// function block for inductive sensor with the option of debouncing + rising and falling edge detection.
FUNCTION_BLOCK FB_InductiveSensor IMPLEMENTS  I_Component
VAR_INPUT
	bSignal			: BOOL;		// Raw input sensor
	tDebounce		: TIME;		// Debounce time
// Interface vars
	sName			: STRING[20];
	bEnable     	: BOOL;
	bStart      	: BOOL;
	bHalt			: BOOL;
	bStop       	: BOOL;
	eMode       	: E_ComponentMode; 		// 0=OFF, 1=AUTO, 2=MANUAL	
END_VAR

VAR_OUTPUT
	bActive			: BOOL;
	bRising			: BOOL;
	bFalling		: BOOL;
// interface vars
	eState			: E_ComponentState;		// 0=READY, 1=BUSY, 2=DONE
	iErrorCode		: INT;
	sStatusText 	: STRING[50];
END_VAR

VAR
	bLastSignal		: BOOL;
	tDebTimer		: TON;
	bSignalStable	: BOOL;
END_VAR

IF bEnable THEN
	IF bLastSignal <> bSignal THEN
		tDebTimer(IN := TRUE, PT := tDebounce);
		eState := E_ComponentState.BUSY;
	ELSE
		tDebTimer(IN := FALSE);
	END_IF
	
	IF tDebTimer.Q THEN
		bSignalStable 	:= bSignal;
		bLastSignal 	:= bSignal;
		eState := E_ComponentState.READY;
	END_IF
	
	bRising		:= (bSignalStable AND NOT bActive);
	bFalling	:= (NOT bSignalStable AND bActive);
	bActive 	:= bSignalStable;
ELSE
	bActive 	:= FALSE;
	bRising		:= FALSE;
	bFalling	:= FALSE;
	tDebTimer(IN := FALSE);
END_IF

METHOD Halt : BOOL
END_METHOD

METHOD Read : BOOL
Read := bSensor;
END_METHOD

METHOD Start : BOOL
END_METHOD

METHOD Stop : BOOL
END_METHOD

END_FUNCTION_BLOCK

(* stored: Version 1.1.0.1, ProductVersion 3.1.4024.15
   POU FB_InductiveSensor: Id {8e7ef9e5-be5c-4d5b-9caf-29f0d28584ab}, SpecialFunc None
   Method Halt: Id {f3238e3e-c657-463e-ba29-1e530a523711}
   Method Read: Id {bddb87fd-a3a6-46c2-996c-bd7bd9b3500c}
   Method Start: Id {332d80dd-0194-4918-b2f7-7e712950268d}
   Method Stop: Id {1e590e11-4492-46f6-8aed-701c371c3bb9} *)
